// Mitsubishi GX Works2 project: KemNghiaDrillV2   PLC: FX3U/FX3UC

// global labels: Global1
VAR_GLOBAL
  XXLimitN AT M8344 : BOOL;
  XXLimitP AT M8343 : BOOL;
  XXBusy AT M8340 : BOOL;
  XXInterruptInverse AT M8347 : BOOL;
  XXPos AT D8340 : DINT;
  XXAccelTime AT D8348 : INT;
  XXDecelTime AT D8349 : INT;
  XXPosView AT D0 : DINT;
  XXTarPos AT D2 : DINT;
  XXFeed AT D4 : DINT;
  XXTarR AT M0 : BOOL;
  XXTarRSkip AT D6 : INT;
  XXManualN AT M1 : BOOL;
  XXManualP AT M2 : BOOL;
  XXOn AT M3 : BOOL;
  XXRun AT M4 : BOOL;
  XXDirection AT M5 : BOOL;
  XXMinI AT X000 : BOOL;
  XXReadyI AT X010 : BOOL;
  XXPulseO AT Y000 : BOOL;
  XXDirectionO AT Y004 : BOOL;
  XXOnO AT Y002 : BOOL;
  YYLimitN AT M8354 : BOOL;
  YYLimitP AT M8353 : BOOL;
  YYBusy AT M8350 : BOOL;
  YYInterruptInverse AT M8357 : BOOL;
  YYPos AT D8350 : DINT;
  YYAccelTime AT D8358 : INT;
  YYDecelTime AT D8359 : INT;
  YYPosView AT D7 : DINT;
  YYTarPos AT D9 : DINT;
  YYFeed AT D11 : DINT;
  YYTarR AT M6 : BOOL;
  YYTarRSkip AT D13 : INT;
  YYManualN AT M7 : BOOL;
  YYManualP AT M8 : BOOL;
  YYOn AT M9 : BOOL;
  YYRun AT M10 : BOOL;
  YYDirection AT M11 : BOOL;
  YYMinI AT X001 : BOOL;
  YYMaxI AT X005 : BOOL;
  YYReadyI AT X011 : BOOL;
  YYPulseO AT Y001 : BOOL;
  YYDirectionO AT Y005 : BOOL;
  YYOnO AT Y006 : BOOL;
  MachineReady AT M12 : BOOL;
  GetOriginDone AT M13 : BOOL;
  DataSynced AT M14 : BOOL;
  Run AT M15 : BOOL;
  RunStop AT M16 : BOOL;
  AccelTime AT D14 : INT;
  DecelTime AT D15 : INT;
  PositionArray AT D1000 : ARRAY [0..7] OF DINT;
  RunState AT D16 : INT;
  RunStateFoilExtract AT D17 : INT;
  RunStateDrill AT D18 : INT;
  RunStateFoilOut AT D19 : INT;
  FoilExtractTopN AT M17 : BOOL;
  FoilExtractTopP AT M18 : BOOL;
  FoilExtractTopNI AT X002 : BOOL;
  FoilExtractTopPI AT X003 : BOOL;
  FoilExtractTop AT M19 : BOOL;
  FoilExtractTopO AT Y003 : BOOL;
  FoilExtractBotN AT M20 : BOOL;
  FoilExtractBotP AT M21 : BOOL;
  FoilExtractBotNI AT X004 : BOOL;
  FoilExtractBotPI AT X006 : BOOL;
  FoilExtractBot AT M22 : BOOL;
  FoilExtractBotO AT Y007 : BOOL;
  Drill AT M23 : BOOL;
  DrillO AT Y010 : BOOL;
  DrillZOriginGetReadyPI AT X007 : BOOL;
  DrillZOriginGetEnable AT M24 : BOOL;
  DrillZOriginGetEnableO AT Y011 : BOOL;
  DrillZOriginGetI AT X012 : BOOL;
  DrillZOrigin AT D20 : DINT;
  DrillZStart AT D22 : DINT;
  DrillZEnd AT D24 : DINT;
  FoilOutN AT M25 : BOOL;
  FoilOutP AT M26 : BOOL;
  FoilOutNI AT X013 : BOOL;
  FoilOutPI AT X014 : BOOL;
  FoilOut AT M27 : BOOL;
  FoilOutO AT Y012 : BOOL;
  AirBurst AT M28 : BOOL;
  AirBurstO AT Y013 : BOOL;
END_VAR

// task Task_01 (event TRUE, interval 0, priority 31): POU_01

PROGRAM POU_01
VAR
  fFall : BOOL;
  fRise : BOOL;
  fTmp : BOOL;
  fRunStateNext : BOOL;
  fRunStateFoilExtractNext : BOOL;
  fRunStateDrillNext : BOOL;
  fRunStateFoilOutNext : BOOL;
  fTurnStepCount : INT;
  fAxisTest : BOOL;
  fAxisDRVIOffset : DINT;
  fStepReady : BOOL;
END_VAR
VAR CONSTANT
  fSectorCount : INT := 1;
END_VAR
VAR
  fAxisDRVIFrequency : DINT;
  fAxisDRVIOffsetBefore : DINT;
  fRunAuto : BOOL;
  fIgnoreDrillTap : BOOL;
END_VAR
SET(M8002, M8336);
MOV(M8002, H01FF, D8336);
RST(M8002, XXInterruptInverse);
ZRST(M8002, RunState, RunStateFoilOut);
SET(M8002, FoilExtractTop);
SET(M8002, FoilExtractBot);
RST(M8002, Drill);
RST(M8002, fAxisTest);
RST(M8002, fIgnoreDrillTap);
RST(M8002, fRunAuto);

(*Set XX to 32768 PPR, from 262144 PPR encoder*)

DMOV(M8002, 150, fAxisDRVIOffset);
DMOV(M8002, 300, fAxisDRVIOffsetBefore); (*offset beforce must larger than offset*)
DMOV(M8002, 300, fAxisDRVIFrequency);

OUT_T(M8000, TC0, 50);
SET(TC0 AND Run AND RunState = 0, fTmp);
RST(fTmp, Run);
MOV(fTmp, 1, RunState);
RST(fTmp, fTmp);
SET(RunStop, fTmp);
RST(fTmp, RunStop);
ZRST(fTmp, RunState, RunStateFoilOut);
ZRST(fTmp, fRunStateFoilOutNext, fRunStateNext);
RST(fTmp, XXRun);
RST(fTmp, XXOn);
RST(fTmp, FoilOut);
RST(fTmp, fRunAuto);
RST(fTmp, fTmp);

INC(fRunStateNext, RunState);
INC(fRunStateFoilExtractNext, RunStateFoilExtract);
INC(fRunStateDrillNext, RunStateDrill);
INC(fRunStateFoilOutNext, RunStateFoilOut);
ZRST(M8000, fRunStateFoilOutNext, fRunStateNext);
DECO(M8000, RunState, 6, M100); DECO(M8000, RunState, 6, M1000); ZRST(NOT XXTarR, M1000, M1063);
DECO(M8000, RunStateFoilExtract, 6, M200);
DECO(M8000, RunStateDrill, 6, M300); DECO(M8000, RunStateDrill, 6, M1300); ZRST(NOT XXTarR, M1300, M1363);
DECO(M8000, RunStateFoilOut, 6, M400);

(*||||||||||*)
(*turn axis on*)
SET(M101 AND NOT XXOn, XXOn);
SET(M101 AND XXReadyI, fRunStateNext);
(*move fast before ddvi*)
DMOVP(M1002, XXPos + PositionArray[0] - fAxisDRVIOffsetBefore, XXTarPos);
SET(M1002, XXRun);
SET(M1002, fRunStateNext);
(*setup ddvi*)
SET(M1003, fRunStateNext);
(*ddvi*)
DDVIT(M104, fAxisDRVIOffset, fAxisDRVIFrequency, XXPulseO, XXDirection);
SET(M104 AND M8029, fRunStateNext);
RST(M104 AND M8029, M104);
(*get origin done*)
RST(M1005, XXPos);
MOV(M1005, 7, RunState);
(*start run*)
RST(M1007, fTurnStepCount);
RST(M1007, XXPos);
MOV(M1007, 14, RunState);
(*move next position*)
DMOV(M1008, PositionArray[fTurnStepCount], XXPos);
SET(M1008, XXRun);
MOV(M1008, 14, RunState);
(*move next position done*)
(*final*) SET(M1014 AND fTurnStepCount = (fSectorCount - 1), fTmp);
(*final*) INC(fTmp, fTurnStepCount);
(*final*) MOV(fTmp, 15, RunState);
(*final*) RST(fTmp, M1014);
(*final*) RST(fTmp, fTmp);
INC(M1014 AND fTurnStepCount < fSectorCount, fTurnStepCount);
(*full turn*) SET(M1014 AND fTurnStepCount >= fSectorCount, fTmp);
(*full turn*) RST(fTmp, fTurnStepCount);
(*full turn*) MOV(fTmp, 2, RunState);
(*full turn*) RST(fTmp, M1014);
(*full turn*) RST(fTmp, fTmp);
MOV(M1014, 15, RunState);
(*process, delay 500ms with TC2 before, why?*)
SET(M1015, AirBurst);
MOV(M1015, 1, RunStateFoilExtract);
MOV(M1015, 1, RunStateDrill);
MOV(M1015, 1, RunStateFoilOut);
SET(M1015, fRunStateNext);
(*wait all done*)
(*test*) OUT_T(M1016, TC3, 5);
(*test*) SET(M1016 AND TC3 AND fAxisTest AND fStepReady, fTmp);
(*test*) RST(fStepReady, fStepReady);
SET(M1016 AND M210 AND M310 AND M410, fTmp);
ZRST(fTmp, RunStateFoilExtract, RunStateFoilOut);
SET(fTmp, fRunStateNext);
RST(fTmp, fTmp);
(*manual step*)
SET(M1017 AND NOT fRunAuto AND Run, fRunStateNext);
SET(M1017 AND fRunAuto, fRunStateNext);
RST(Run, Run);
(**)
SET(M1018 AND fSectorCount = 1, fTmp);
MOV(fTmp, 2, RunState);
RST(fTmp, M1018);
RST(fTmp, fTmp);
SET(M1018 AND fTurnStepCount = fSectorCount, fTmp);
MOV(M1018 AND NOT fTmp, 8, RunState);
MOV(M1018 AND fTmp, 14, RunState);
RST(fTmp, fTmp);
(**)
(*||||||||||*)
(*||||||||||FoilExtract*)
(*not ready, top and bot forward*)
SET(M201 AND NOT FoilExtractTopP, FoilExtractTop);
SET(M201 AND NOT FoilExtractBotP, FoilExtractBot);
RST(M201 AND NOT (FoilExtractTopP OR FoilExtractBotP), M201);
(*ready, bot back*)
RST(M201, FoilExtractBot);
SET(M201, fRunStateFoilExtractNext);
(*bot back done, bot forward*)
RST(M202 AND NOT FoilExtractBotN, M202);
SET(M202, FoilExtractBot);
SET(M202, fRunStateFoilExtractNext);
(*bot forward done, top back*)
OUT_T(M203, TC50, 5);
SET(M203 AND TC50 AND FoilExtractBotP, fTmp);
RST(fTmp, FoilExtractTop);
SET(fTmp, fRunStateFoilExtractNext);
RST(fTmp, fTmp);
(*top back done, top forward*)
RST(M204 AND NOT FoilExtractTopN, M204);
SET(M204, FoilExtractTop);
SET(M204, fRunStateFoilExtractNext);
(*top forward done, end*)
MOV(M205 AND FoilExtractTopP, 10, RunStateFoilExtract);
(*||||||||||*)
(*||||||||||Drill*)
(**)
MOV(M301 AND fIgnoreDrillTap, 10, RunStateDrill);
SET(M301 AND NOT fIgnoreDrillTap, fRunStateDrillNext);
(**)
SET(M302 AND YYMinI, fRunStateDrillNext);
(*||||||||||*)
(*||||||||||FoilOut*)
(**)
RST(M401 AND NOT FoilOutN, FoilOut);
SET(M401 AND FoilOutN, fRunStateFoilOutNext);
(**)
SET(M402, FoilOut);
SET(M402, fRunStateFoilOutNext);
(**)
RST(M403 AND FoilOutP, FoilOut);
SET(M403 AND FoilOutP, fRunStateFoilOutNext);
(*down done, end*)
MOV(M404 AND FoilOutN, 10, RunStateFoilOut);
(*||||||||||*)

(*||||||||||*)
RST(XXRun AND XXTarPos = XXPos, XXRun);
DDRVA(XXRun, XXTarPos, XXFeed, XXPulseO, XXDirection);
RST(M8029, XXRun);
OUT(XXDirection, XXDirectionO);
INC(NOT XXRun AND NOT XXBusy AND XXTarRSkip < 5, XXTarRSkip);
RST(XXRun, XXTarRSkip);
OUT(XXTarRSkip >= 5, XXTarR);
(*||||||||||*)
(*||||||||||*)
RST(YYRun AND YYTarPos = YYPos, YYRun);
DDRVA(YYRun, YYTarPos, YYFeed, YYPulseO, YYDirection);
RST(M8029, YYRun);
OUT(YYDirection, YYDirectionO);
INC(NOT YYRun AND NOT YYBusy AND YYTarRSkip < 5, YYTarRSkip);
RST(YYRun, YYTarRSkip);
OUT(YYTarRSkip >= 5, YYTarR);
(*||||||||||*)

(**)
OUT_T(NOT FoilExtractTop, TC10, 10); SET(TC10, FoilExtractTopN); RST(TC10, FoilExtractTopP);
OUT_T(FoilExtractTop, TC11, 3); SET(TC11, FoilExtractTopP); RST(TC11, FoilExtractTopN);
(**)
OUT_T(NOT FoilExtractBot, TC12, 10); SET(TC12, FoilExtractBotN); RST(TC12, FoilExtractBotP);
OUT_T(FoilExtractBot, TC13, 3); SET(TC13, FoilExtractBotP); RST(TC13, FoilExtractBotN);
(**)

(**)
OUT_T(FoilOutNI, TC18, 3); SET(TC18, FoilOutN); RST(TC18, FoilOutP);
OUT_T(FoilOutPI, TC19, 3); SET(TC19, FoilOutP); RST(TC19, FoilOutN);
(**)

(*Output*)
OUT_T(AirBurst, TC20, 10); RST(TC20, AirBurst);
(**)
OUT(XXOn, XXOnO);
OUT(YYOn, YYOnO);
OUT(NOT FoilExtractTop, FoilExtractTopO);
OUT(NOT FoilExtractBot, FoilExtractBotO);
OUT(Drill, DrillO);
OUT(FoilOut, FoilOutO);
OUT(AirBurst, AirBurstO);
END_PROGRAM
